# EPICS autosave request: ipApp/Db/deviceCmdReply_settings.req
file scalcout_settings.req P=$(P)cmdReply$(N)_formatCmd
file asynRecord_settings.req P=$(P)cmdReply$(N)_do_IO
file scalcout_settings.req P=$(P)cmdReply$(N)_parseReply
